// TIA Portal project "双通道流水线" (V16)

(* hardware
DEVICE "HMI_1"  KTP700 Basic PN
   slot 0: "HMI_1"  KTP700 Basic PN  6AV2 123-2GB03-0AX0  16.0.0.0
   slot 1: "HMI_RT_1"  KTP700 Basic PN  6AV2 123-2GB03-0AX0  16.0.0.0
   slot 5: "HMI_1.IE_CP_1"  PROFINET Interface  16.0.0.0
      slot 1: "PROFINET Interface_1"  PROFINET Interface
         slot 1: "Port_1"  Port
DEVICE "S7-1200 station_1"  S7-1200 Station
   slot 0: "Rack_0"  S7-1200 Rack  Rack  V1.0
   slot 1: "PLC_1"  CPU 1214C DC/DC/Rly  6ES7 214-1HG40-0XB0  V4.4
*)

// ===== PLC "PLC_1"  CPU 1214C DC/DC/Rly =====

VAR_GLOBAL   // PLC tag table "中间变量"
   "中间变量1" AT %M0.0 : Bool;
   "中间变量2" AT %M0.1 : Bool;
   "中间变量3" AT %M0.2 : Bool;
   "中间变量4" AT %M0.3 : Bool;
   "中间变量5" AT %M0.4 : Bool;
   "中间变量6" AT %M0.5 : Bool;
   "中间变量7" AT %M0.6 : Bool;
   "中间变量8" AT %M0.7 : Bool;
   "中间变量9" AT %M1.0 : Bool;
   "中间变量10" AT %M1.1 : Bool;
   "启动标志位1" AT %M1.2 : Bool;
   "启动标志位2" AT %M1.3 : Bool;
END_VAR

VAR_GLOBAL   // PLC tag table "io表"
   "传感器1" AT %I2.0 : Bool;
   "传感器2" AT %I2.1 : Bool;
   "电容传感器2" AT %I2.3 : Bool;
   "显示屏传感器" AT %I2.4 : Bool;
   "启动按钮" AT %I2.5 : Bool;
   "复位按钮" AT %I2.6 : Bool;
   "停止按钮" AT %I2.7 : Bool;
   "急停" AT %I3.0 : Bool;
   "自动模式" AT %I3.1 : Bool;
   "FACTORY I/O (Running)" AT %I3.3 : Bool;
   "传送带1" AT %Q2.0 : Bool;
   "正转1" AT %Q2.1 : Bool;
   "反转1" AT %Q2.2 : Bool;
   "上升右行1" AT %Q2.3 : Bool;
   "上升左行1" AT %Q2.4 : Bool;
   "传送带2" AT %Q2.5 : Bool;
   "正转2" AT %Q2.6 : Bool;
   "反转2" AT %Q2.7 : Bool;
   "上升右行2" AT %Q3.0 : Bool;
   "上升左行2" AT %Q3.1 : Bool;
   "传送带3" AT %Q3.2 : Bool;
   "绿色" AT %Q3.3 : Bool;
   "黄色" AT %Q3.4 : Bool;
   "红色" AT %Q3.5 : Bool;
   "显示屏" AT %QD30 : DInt;
   "电容式传感器1" AT %I2.2 : Bool;
   "手动模式" AT %I3.2 : Bool;
   "上料端1" AT %Q3.6 : Bool;
   "上料端2" AT %Q3.7 : Bool;
END_VAR

DATA_BLOCK "主程序DB块"   // DB1
{ S7_Optimized_Access := 'TRUE' }
VERSION : 0.1
   VAR
      运行模式 : DInt;
   END_VAR
BEGIN
END_DATA_BLOCK

// folder: 01-核心程序块

DATA_BLOCK "核心程序块_DB"   // DB2
{ S7_Optimized_Access := 'TRUE' }
VERSION : 0.1
// stored: InstanceOfName 核心程序块
"核心程序块"
BEGIN
END_DATA_BLOCK

// folder: 02-自动模式

DATA_BLOCK "自动运行_DB"   // DB3
{ S7_Optimized_Access := 'TRUE' }
VERSION : 0.1
// stored: InstanceOfName 自动运行
"自动运行"
BEGIN
END_DATA_BLOCK

// folder: 03-手动模式

DATA_BLOCK "手动运行_DB"   // DB4
{ S7_Optimized_Access := 'TRUE' }
VERSION : 0.1
// stored: InstanceOfName 手动运行
"手动运行"
BEGIN
END_DATA_BLOCK

// folder: 04-系统停止

DATA_BLOCK "系统停止_DB"   // DB5
{ S7_Optimized_Access := 'TRUE' }
VERSION : 0.1
// stored: InstanceOfName 系统停止
"系统停止"
BEGIN
END_DATA_BLOCK

// folder: (top level)

FUNCTION "MHJ-PLC-Lab-Function-S71200" : Void   // FC9000, SCL
{ S7_Optimized_Access := 'TRUE' }
VERSION : 0.1
   VAR_TEMP
      rdTimeReturn : Int;
      outputTime : DTL;
      SyncVal : Byte;
      forVal : Int;
      forVal_2 : Int;
      Value : Byte;
   END_VAR
   VAR CONSTANT
      CompVal : Byte := 16#34;
      Value_01 : Byte := 16#11;
      Value_01_DW : DWord := 16#A165_D992;
      Value_02_DW : DWord := 16#58BE_4401;
   END_VAR
BEGIN

   #Value:=PEEK(area := 16#82,
        dbNumber := 0,
        byteOffset := 511);
   #Value := #Value + 1;

   POKE(area := 16#82,
        dbNumber := 0,
        byteOffset := 511,
        value := #Value);

   POKE(area:=16#81,
        dbNumber:=0,
        byteOffset:=1016,
        value:=#Value_01_DW);
   POKE(area := 16#81,
        dbNumber := 0,
        byteOffset := 1020,
        value := #Value_02_DW);

   POKE(area := 16#81,
        dbNumber := 0,
        byteOffset := 511,
        value := B#16#00);

   FOR #forVal := 0 TO 120 DO
       FOR #forVal_2:=0 TO 10 DO
           #rdTimeReturn:=RD_SYS_T(#outputTime);
           #rdTimeReturn := WR_SYS_T(#outputTime);
           #rdTimeReturn := RD_SYS_T(#outputTime);
           #rdTimeReturn := WR_SYS_T(#outputTime);
       END_FOR;
       #SyncVal:= PEEK(area := 16#81,
                      dbNumber := 0,
                      byteOffset := 511);
       IF #SyncVal = #CompVal THEN
          GOTO M_1;
       END_IF;
   END_FOR;
   RETURN;

   M_1:
   POKE(area := 16#81,
        dbNumber := 0,
        byteOffset := 511,
        value := B#16#0);
END_FUNCTION

ORGANIZATION_BLOCK "Main"   // OB1, LAD, ProgramCycle
TITLE = "Main Program Sweep (Cycle)"
{ S7_Optimized_Access := 'TRUE' }
VERSION : 0.1
   VAR_INPUT
      Initial_Call : Bool;   // Initial call of this OB
      Remanence : Bool;   // =True, if remanent data are available
   END_VAR
BEGIN

REGION Network 1
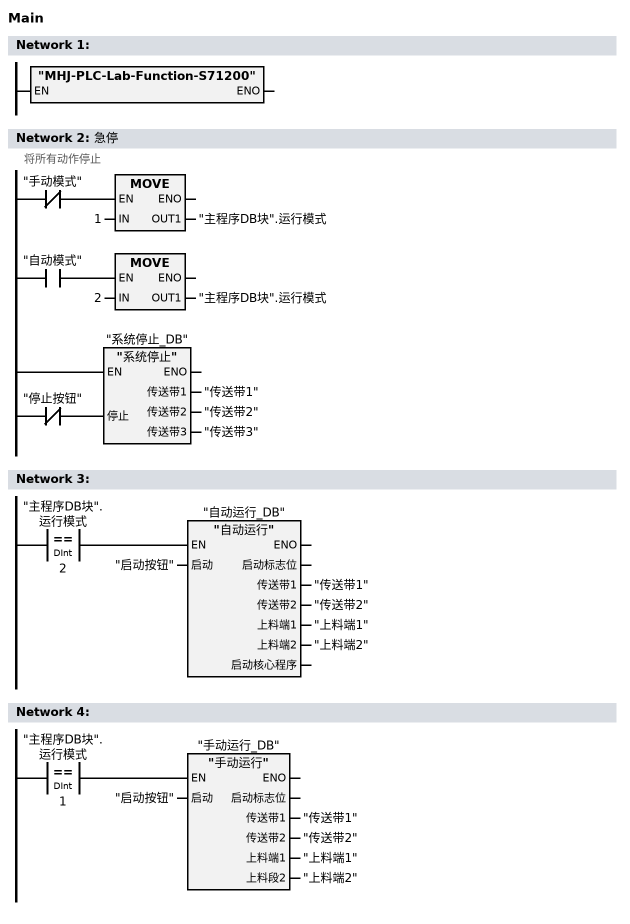
   RUNG wire#powerrail
      "MHJ-PLC-Lab-Function-S71200"()
   END_RUNG
   // the same network as SCL:
   "MHJ-PLC-Lab-Function-S71200"();
END_REGION

REGION Network 2: 急停
   // 将所有动作停止
   RUNG wire#powerrail
      I_Contact( "手动模式" )
      Move(in := 1, out1 => "主程序DB块".运行模式)
   END_RUNG
   RUNG wire#powerrail
      Contact( "自动模式" )
      Move(in := 2, out1 => "主程序DB块".运行模式)
   END_RUNG
   RUNG wire#powerrail
      "系统停止_DB"(停止 := wire#w1, 传送带1 => "传送带1", 传送带2 => "传送带2", 传送带3 => "传送带3")
   END_RUNG
   RUNG wire#powerrail
      I_Contact( "停止按钮" )
   END_RUNG wire#w1
   // the same network as SCL:
   IF NOT "手动模式" THEN "主程序DB块".运行模式 := 1; END_IF;
   IF "自动模式" THEN "主程序DB块".运行模式 := 2; END_IF;
   "系统停止_DB"(停止 := NOT "停止按钮", 传送带1 => "传送带1", 传送带2 => "传送带2", 传送带3 => "传送带3");   // "系统停止"
END_REGION

REGION Network 3
   RUNG wire#powerrail
      { S7_Templates := "SrcType := DInt" } EQ_Contact(in1 := "主程序DB块".运行模式, in2 := 2)
      "自动运行_DB"(启动 := "启动按钮", 启动标志位 =>, 传送带1 => "传送带1", 传送带2 => "传送带2", 上料端1 => "上料端1", 上料端2 => "上料端2", 启动核心程序 =>)
   END_RUNG
   // the same network as SCL:
   IF "主程序DB块".运行模式 = 2 THEN
       "自动运行_DB"(启动 := "启动按钮", 传送带1 => "传送带1", 传送带2 => "传送带2", 上料端1 => "上料端1", 上料端2 => "上料端2");   // "自动运行"
   END_IF;
END_REGION

REGION Network 4
   RUNG wire#powerrail
      { S7_Templates := "SrcType := DInt" } EQ_Contact(in1 := "主程序DB块".运行模式, in2 := 1)
      "手动运行_DB"(启动 := "启动按钮", 启动标志位 =>, 传送带1 => "传送带1", 传送带2 => "传送带2", 上料端1 => "上料端1", 上料段2 => "上料端2")
   END_RUNG
   // the same network as SCL:
   IF "主程序DB块".运行模式 = 1 THEN
       "手动运行_DB"(启动 := "启动按钮", 传送带1 => "传送带1", 传送带2 => "传送带2", 上料端1 => "上料端1", 上料段2 => "上料端2");   // "手动运行"
   END_IF;
END_REGION
END_ORGANIZATION_BLOCK

// folder: 01-核心程序块

FUNCTION_BLOCK "核心程序块"   // FB1, LAD
{ S7_Optimized_Access := 'TRUE' }
VERSION : 0.1
   VAR_INPUT
      传感器1 : Bool;
      传感器2 : Bool;
      电容传感器1 : Bool;
      电容传感器2 : Bool;
      显示屏传感 : Bool;
      启动 : Bool;
   END_VAR
   VAR_OUTPUT
      正转1 : Bool;
      正转2 : Bool;
      上升左行1 : Bool;
      上升左行2 : Bool;
      传送带1 : Bool;
      传送带2 : Bool;
      传送带3 : Bool;
      启动标志位 : Bool;
      显示屏 : DInt;
   END_VAR
   VAR
      中间变量1 : Bool;
      中间变量2 : Bool;
      中间变量3 : Bool;
      中间变量4 : Bool;
      中间变量5 : Bool;
      中间变量6 : Bool;
      中间变量7 : Bool;
      中间变量8 : Bool;
      恢复启动函数 : DInt;
   END_VAR
   VAR_TEMP   // added for the SCL form of the ladder/FBD networks
      _w1 : Bool;
      _w2 : Bool;
      _w3 : Bool;
      _w4 : Bool;
   END_VAR
BEGIN

REGION Network 1
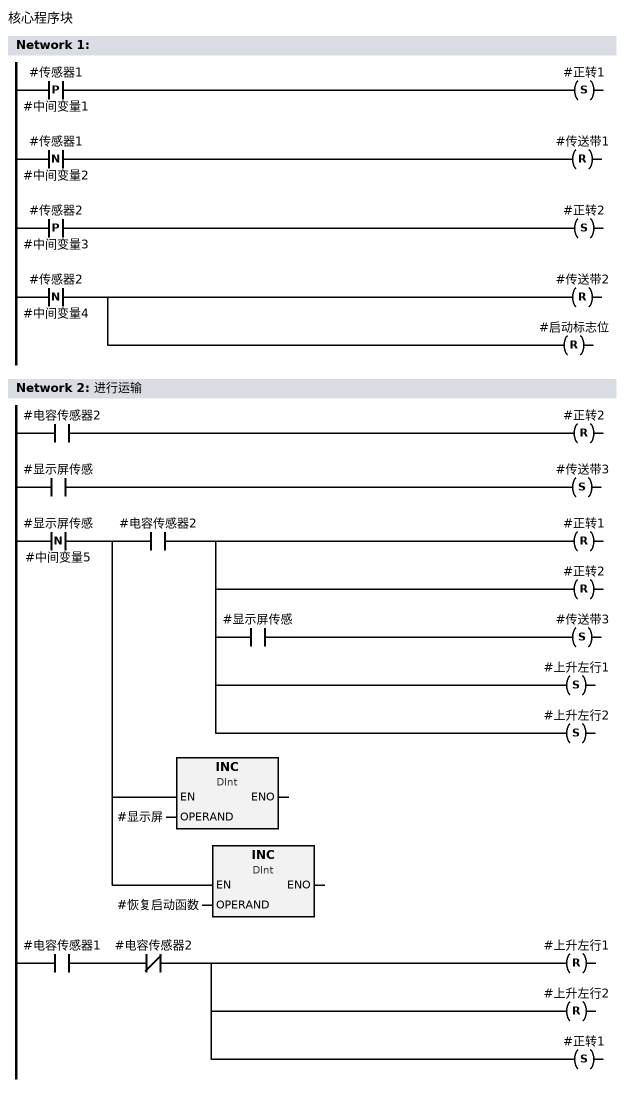
   RUNG wire#powerrail
      P_Contact(operand := #传感器1, bit := #中间变量1)
      S_Coil( #正转1 )
   END_RUNG
   RUNG wire#powerrail
      N_Contact(operand := #传感器1, bit := #中间变量2)
      R_Coil( #传送带1 )
   END_RUNG
   RUNG wire#powerrail
      P_Contact(operand := #传感器2, bit := #中间变量3)
      S_Coil( #正转2 )
   END_RUNG
   RUNG wire#powerrail
      N_Contact(operand := #传感器2, bit := #中间变量4)
      wire#w1
      R_Coil( #传送带2 )
   END_RUNG
   RUNG wire#w1
      R_Coil( #启动标志位 )
   END_RUNG
   // the same network as SCL:
   #_w1 := #传感器1 AND NOT #中间变量1;   // rising edge of #传感器1
   #中间变量1 := #传感器1;
   IF #_w1 THEN #正转1 := TRUE; END_IF;
   #_w2 := NOT #传感器1 AND #中间变量2;   // falling edge of #传感器1
   #中间变量2 := #传感器1;
   IF #_w2 THEN #传送带1 := FALSE; END_IF;
   #_w3 := #传感器2 AND NOT #中间变量3;   // rising edge of #传感器2
   #中间变量3 := #传感器2;
   IF #_w3 THEN #正转2 := TRUE; END_IF;
   #_w4 := NOT #传感器2 AND #中间变量4;   // falling edge of #传感器2
   #中间变量4 := #传感器2;
   IF #_w4 THEN
       #传送带2 := FALSE;
       #启动标志位 := FALSE;
   END_IF;
END_REGION

REGION Network 2: 进行运输
   RUNG wire#powerrail
      Contact( #电容传感器2 )
      R_Coil( #正转2 )
   END_RUNG
   RUNG wire#powerrail
      Contact( #显示屏传感 )
      S_Coil( #传送带3 )
   END_RUNG
   RUNG wire#powerrail
      N_Contact(operand := #显示屏传感, bit := #中间变量5)
      wire#w1
      Contact( #电容传感器2 )
      wire#w2
      R_Coil( #正转1 )
   END_RUNG
   RUNG wire#w2
      R_Coil( #正转2 )
   END_RUNG
   RUNG wire#w2
      Contact( #显示屏传感 )
      S_Coil( #传送带3 )
   END_RUNG
   RUNG wire#w2
      S_Coil( #上升左行1 )
   END_RUNG
   RUNG wire#w2
      S_Coil( #上升左行2 )
   END_RUNG
   RUNG wire#w1
      { S7_Templates := "DestType := DInt" } Inc( #显示屏 )
   END_RUNG
   RUNG wire#w1
      { S7_Templates := "DestType := DInt" } Inc( #恢复启动函数 )
   END_RUNG
   RUNG wire#powerrail
      Contact( #电容传感器1 )
      I_Contact( #电容传感器2 )
      wire#w3
      R_Coil( #上升左行1 )
   END_RUNG
   RUNG wire#w3
      R_Coil( #上升左行2 )
   END_RUNG
   RUNG wire#w3
      S_Coil( #正转1 )
   END_RUNG
   // the same network as SCL:
   IF #电容传感器2 THEN #正转2 := FALSE; END_IF;
   IF #显示屏传感 THEN #传送带3 := TRUE; END_IF;
   #_w1 := NOT #显示屏传感 AND #中间变量5;   // falling edge of #显示屏传感
   #中间变量5 := #显示屏传感;
   #_w2 := #_w1 AND #电容传感器2;
   IF #_w2 THEN
       #正转1 := FALSE;
       #正转2 := FALSE;
   END_IF;
   IF #_w2 AND #显示屏传感 THEN #传送带3 := TRUE; END_IF;
   IF #_w2 THEN
       #上升左行1 := TRUE;
       #上升左行2 := TRUE;
   END_IF;
   IF #_w1 THEN
       #显示屏 := #显示屏 + 1;
       #恢复启动函数 := #恢复启动函数 + 1;
   END_IF;
   IF #电容传感器1 AND NOT #电容传感器2 THEN
       #上升左行1 := FALSE;
       #上升左行2 := FALSE;
       #正转1 := TRUE;
   END_IF;
END_REGION
END_FUNCTION_BLOCK

// folder: 02-自动模式

FUNCTION_BLOCK "自动运行"   // FB2, LAD
{ S7_Optimized_Access := 'TRUE' }
VERSION : 0.1
   VAR_INPUT
      启动 : Bool;
   END_VAR
   VAR_OUTPUT
      启动标志位 : Bool;
      传送带1 : Bool;
      传送带2 : Bool;
      上料端1 : Bool;
      上料端2 : Bool;
      启动核心程序 : Bool;
   END_VAR
   VAR_TEMP   // added for the SCL form of the ladder/FBD networks
      _w1 : Bool;
   END_VAR
BEGIN

REGION Network 1: 启动
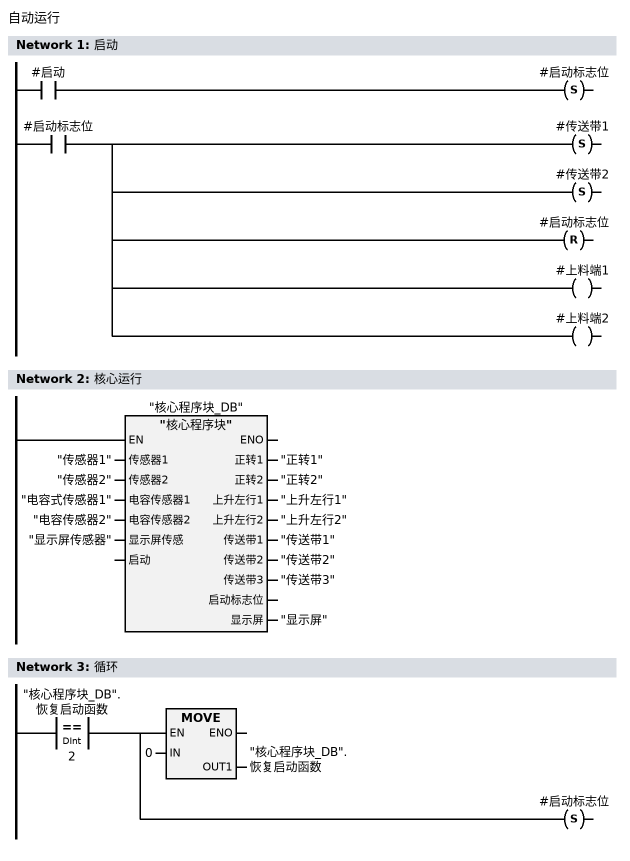
   RUNG wire#powerrail
      Contact( #启动 )
      S_Coil( #启动标志位 )
   END_RUNG
   RUNG wire#powerrail
      Contact( #启动标志位 )
      wire#w1
      S_Coil( #传送带1 )
   END_RUNG
   RUNG wire#w1
      S_Coil( #传送带2 )
   END_RUNG
   RUNG wire#w1
      R_Coil( #启动标志位 )
   END_RUNG
   RUNG wire#w1
      Coil( #上料端1 )
   END_RUNG
   RUNG wire#w1
      Coil( #上料端2 )
   END_RUNG
   // the same network as SCL:
   IF #启动 THEN #启动标志位 := TRUE; END_IF;
   IF #启动标志位 THEN
       #传送带1 := TRUE;
       #传送带2 := TRUE;
   END_IF;
   #_w1 := #启动标志位;
   IF #_w1 THEN #启动标志位 := FALSE; END_IF;
   #上料端1 := #_w1;
   #上料端2 := #_w1;
END_REGION

REGION Network 2: 核心运行
   RUNG wire#powerrail
      "核心程序块_DB"(传感器1 := "传感器1", 传感器2 := "传感器2", 电容传感器1 := "电容式传感器1", 电容传感器2 := "电容传感器2", 显示屏传感 := "显示屏传感器", 启动 :=, 正转1 => "正转1", 正转2 => "正转2", 上升左行1 => "上升左行1", 上升左行2 => "上升左行2", 传送带1 => "传送带1", 传送带2 => "传送带2", 传送带3 => "传送带3", 启动标志位 =>, 显示屏 => "显示屏")
   END_RUNG
   // the same network as SCL:
   "核心程序块_DB"(传感器1 := "传感器1",   // "核心程序块"
              传感器2 := "传感器2",
              电容传感器1 := "电容式传感器1",
              电容传感器2 := "电容传感器2",
              显示屏传感 := "显示屏传感器",
              正转1 => "正转1",
              正转2 => "正转2",
              上升左行1 => "上升左行1",
              上升左行2 => "上升左行2",
              传送带1 => "传送带1",
              传送带2 => "传送带2",
              传送带3 => "传送带3",
              显示屏 => "显示屏");
END_REGION

REGION Network 3: 循环
   RUNG wire#powerrail
      { S7_Templates := "SrcType := DInt" } EQ_Contact(in1 := "核心程序块_DB".恢复启动函数, in2 := 2)
      wire#w1
      Move(in := 0, out1 => "核心程序块_DB".恢复启动函数)
   END_RUNG
   RUNG wire#w1
      S_Coil( #启动标志位 )
   END_RUNG
   // the same network as SCL:
   #_w1 := "核心程序块_DB".恢复启动函数 = 2;
   IF #_w1 THEN
       "核心程序块_DB".恢复启动函数 := 0;
       #启动标志位 := TRUE;
   END_IF;
END_REGION
END_FUNCTION_BLOCK

// folder: 03-手动模式

FUNCTION_BLOCK "手动运行"   // FB3, LAD
{ S7_Optimized_Access := 'TRUE' }
VERSION : 0.1
   VAR_INPUT
      启动 : Bool;
   END_VAR
   VAR_OUTPUT
      启动标志位 : Bool;
      传送带1 : Bool;
      传送带2 : Bool;
      上料端1 : Bool;
      上料段2 : Bool;
   END_VAR
   VAR_TEMP   // added for the SCL form of the ladder/FBD networks
      _w1 : Bool;
   END_VAR
BEGIN

REGION Network 1
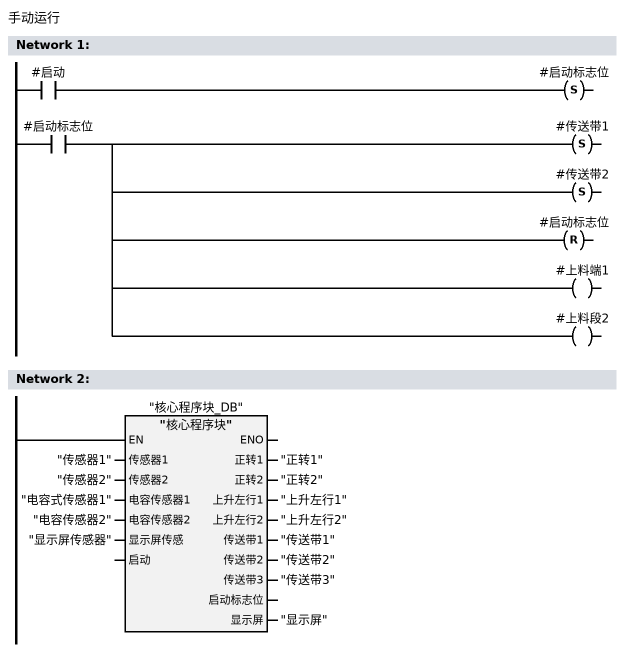
   RUNG wire#powerrail
      Contact( #启动 )
      S_Coil( #启动标志位 )
   END_RUNG
   RUNG wire#powerrail
      Contact( #启动标志位 )
      wire#w1
      S_Coil( #传送带1 )
   END_RUNG
   RUNG wire#w1
      S_Coil( #传送带2 )
   END_RUNG
   RUNG wire#w1
      R_Coil( #启动标志位 )
   END_RUNG
   RUNG wire#w1
      Coil( #上料端1 )
   END_RUNG
   RUNG wire#w1
      Coil( #上料段2 )
   END_RUNG
   // the same network as SCL:
   IF #启动 THEN #启动标志位 := TRUE; END_IF;
   IF #启动标志位 THEN
       #传送带1 := TRUE;
       #传送带2 := TRUE;
   END_IF;
   #_w1 := #启动标志位;
   IF #_w1 THEN #启动标志位 := FALSE; END_IF;
   #上料端1 := #_w1;
   #上料段2 := #_w1;
END_REGION

REGION Network 2
   RUNG wire#powerrail
      "核心程序块_DB"(传感器1 := "传感器1", 传感器2 := "传感器2", 电容传感器1 := "电容式传感器1", 电容传感器2 := "电容传感器2", 显示屏传感 := "显示屏传感器", 启动 :=, 正转1 => "正转1", 正转2 => "正转2", 上升左行1 => "上升左行1", 上升左行2 => "上升左行2", 传送带1 => "传送带1", 传送带2 => "传送带2", 传送带3 => "传送带3", 启动标志位 =>, 显示屏 => "显示屏")
   END_RUNG
   // the same network as SCL:
   "核心程序块_DB"(传感器1 := "传感器1",   // "核心程序块"
              传感器2 := "传感器2",
              电容传感器1 := "电容式传感器1",
              电容传感器2 := "电容传感器2",
              显示屏传感 := "显示屏传感器",
              正转1 => "正转1",
              正转2 => "正转2",
              上升左行1 => "上升左行1",
              上升左行2 => "上升左行2",
              传送带1 => "传送带1",
              传送带2 => "传送带2",
              传送带3 => "传送带3",
              显示屏 => "显示屏");
END_REGION
END_FUNCTION_BLOCK

// folder: 04-系统停止

FUNCTION_BLOCK "系统停止"   // FB4, LAD
{ S7_Optimized_Access := 'TRUE' }
VERSION : 0.1
   VAR_INPUT
      停止 : Bool;
   END_VAR
   VAR_OUTPUT
      传送带1 : Bool;
      传送带2 : Bool;
      传送带3 : Bool;
   END_VAR
BEGIN

REGION Network 1
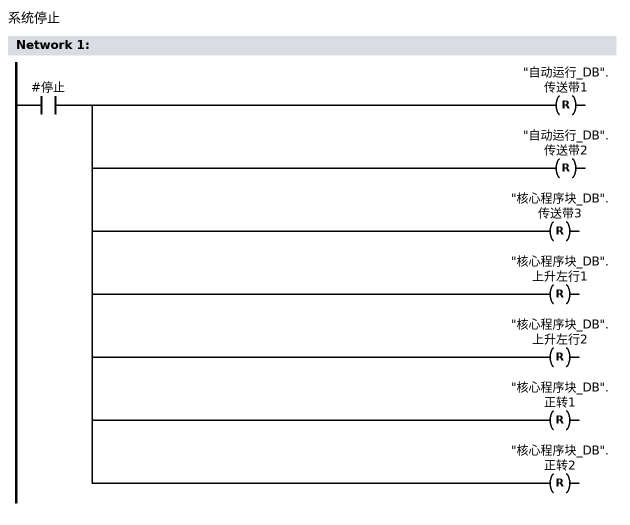
   RUNG wire#powerrail
      Contact( #停止 )
      wire#w1
      R_Coil( "自动运行_DB".传送带1 )
   END_RUNG
   RUNG wire#w1
      R_Coil( "自动运行_DB".传送带2 )
   END_RUNG
   RUNG wire#w1
      R_Coil( "核心程序块_DB".传送带3 )
   END_RUNG
   RUNG wire#w1
      R_Coil( "核心程序块_DB".上升左行1 )
   END_RUNG
   RUNG wire#w1
      R_Coil( "核心程序块_DB".上升左行2 )
   END_RUNG
   RUNG wire#w1
      R_Coil( "核心程序块_DB".正转1 )
   END_RUNG
   RUNG wire#w1
      R_Coil( "核心程序块_DB".正转2 )
   END_RUNG
   // the same network as SCL:
   IF #停止 THEN
       "自动运行_DB".传送带1 := FALSE;
       "自动运行_DB".传送带2 := FALSE;
       "核心程序块_DB".传送带3 := FALSE;
       "核心程序块_DB".上升左行1 := FALSE;
       "核心程序块_DB".上升左行2 := FALSE;
       "核心程序块_DB".正转1 := FALSE;
       "核心程序块_DB".正转2 := FALSE;
   END_IF;
END_REGION
END_FUNCTION_BLOCK

(* ===== HMI "HMI_RT_1" =====
system functions are stored by id; their names below are inferred from use
connection "HMI_连接_1": ETHERNET, SMART_S7_1200_OMS

HMI tags "默认变量表"
   "Tag_ScreenNumber" : UInt, internal

Template "模板_1" 800x480
   Button "退出" at 714,429 size 71x50; TextOff '退出'; PictureOff "ExitRuntime_KTP700_Basic_PN_TR"; PictureOn "ExitRuntime_KTP700_Basic_PN_TR"
      on Release: StopRuntime(0)
   Button "Template_Button" at 614,429 size 71x50; TextOff 'Text'
   Button "Template_Button_1" at 514,429 size 71x50; TextOff 'Text'
   Button "Template_Button_2" at 414,429 size 71x50; TextOff 'Text'
   Button "Template_Button_3" at 314,429 size 71x50; TextOff 'Text'
   Button "Template_Button_4" at 214,429 size 71x50; TextOff 'Text'
   Button "Template_Button_5" at 114,429 size 71x50; TextOff 'Text'
   Button "起始画面" at 14,429 size 71x50; TextOff '起始画面'; PictureOff "NavigateHome_KTP700_Basic_PN_TR"; PictureOn "NavigateHome_KTP700_Basic_PN_TR"
      on Release: ActivateScreen("根画面", 0)
   SymbolicIOField "Symbolic_IO_Field_Screen" at 93,9 size 600x33; TextOff '0'; TextOn '1'; TextList "TextList_ScreenNames"
      ProcessValue <- "Tag_ScreenNumber"
      on Change: ActivateScreenByNumber("Tag_ScreenNumber", 0)
   DateTimeField "HmiScreenItemData" at 695,25 size 105x25
   DateTimeField "HmiScreenItemData_1" at 695,0 size 105x25
   GraphicView "Logo" at 0,0 size 91x51; Picture "HMI_1 的 Logo"

screen "根画面" 800x480, template "模板_1"
   on GenerateScreen: SetTag("Tag_ScreenNumber", 1)
   TextField "HmiScreenItemData" at 80,225 size 640x25; Text '欢迎进入 HMI_1 (KTP700 Basic+ PN)！'
*)